// TIA Portal project "Bloques_y_Lenguajes" (V15)

(* hardware
DEVICE "S7-1200 station_1"  S7-1200 Station
   slot 0: "Rack_0"  S7-1200 Rack  Rack  V1.0
   slot 1: "PLC_1"  CPU 1215C DC/DC/DC  6ES7 215-1AG40-0XB0  V4.2
*)

// ===== PLC "PLC_1"  CPU 1215C DC/DC/DC =====

VAR_GLOBAL   // PLC tag table "Tabla de variables estándar"
   "MarcaTemperatura" AT %MD0 : Real;
   "Temperatura" AT %MD4 : Real;
   "Probabilidad_Temperatura" AT %MD8 : Real;
   "Presion" AT %MD12 : Real;
   "Probabilidad_Presion" AT %MD16 : Real;
   "Indicador_anomalia" AT %M20.0 : Bool;
   "Epsilon" AT %MD22 : Real;
   "Probabilidad_combinada" AT %MD26 : Real;
END_VAR

DATA_BLOCK "Variables1"   // DB1
{ S7_Optimized_Access := 'TRUE' }
VERSION : 0.1
   VAR
      Temperatura : Array[0..3600] of Real;
   END_VAR
   VAR RETAIN
      Puntero : Int := 1;
   END_VAR
   VAR
      Inyectora : Struct
         Temperatura : Struct
            Zona1 : Real;
            Zona2 : Real;
            Zona3 : Real;
            Zona4 : Real;
         END_STRUCT;
         Estado : Bool;
         Alarma : Bool;
      END_STRUCT;
   END_VAR
BEGIN
   Temperatura[5] := 235.87;
END_DATA_BLOCK

FUNCTION "Bloque_SCL" : Void   // FC1, SCL
{ S7_Optimized_Access := 'TRUE' }
VERSION : 0.1
BEGIN
   "MarcaTemperatura" := "Variables1".Temperatura["Variables1".Puntero];
END_FUNCTION

FUNCTION "Calacular_probabilidad_normal_temp" : Void   // FC2, SCL
{ S7_Optimized_Access := 'TRUE' }
VERSION : 0.1
   VAR_INPUT
      Media : Real;
      Desviacion_estandar : Real;
      Nuevo_Dato : Real;
   END_VAR
   VAR_OUTPUT
      Probabilidad : Real;
   END_VAR
   VAR CONSTANT
      Pi : Real := 3.1416;
   END_VAR
BEGIN
   #Probabilidad := EXP(-0.5 * SQR((#Nuevo_Dato - #Media) / #Desviacion_estandar))/((#Desviacion_estandar * SQRT(2.0*#Pi)));
END_FUNCTION

FUNCTION "Detector_de_anamolia" : Void   // FC3, SCL
{ S7_Optimized_Access := 'TRUE' }
VERSION : 0.1
   VAR_INPUT
      Probabilidad1 : Real;
      Probabilidad2 : Real;
      Epsilon : Real;
   END_VAR
   VAR_OUTPUT
      Indicacion_anomalia : Bool;
      "V alorProbabilidad_combinada" : Real;
   END_VAR
BEGIN
   IF #Probabilidad1 * #Probabilidad2 > #Epsilon  THEN
       #Indicacion_anomalia:=FALSE
       ;
   END_IF;

   IF #Probabilidad1 * #Probabilidad2 < #Epsilon THEN
       #Indicacion_anomalia:=TRUE
       ;
   END_IF;

   #"V alorProbabilidad_combinada" := #Probabilidad1 * #Probabilidad2;
END_FUNCTION

FUNCTION "Calcular_probabilidad_normal_presion" : Void   // FC4, SCL
{ S7_Optimized_Access := 'TRUE' }
VERSION : 0.1
   VAR_INPUT
      Media1 : Real;
      Desviacion_estandar1 : Real;
      Nuevo_Dato1 : Real;
   END_VAR
   VAR_OUTPUT
      Probabilidad1 : Real;
   END_VAR
   VAR CONSTANT
      Pi1 : Real := 3.1416;
   END_VAR
BEGIN
   #Probabilidad1 := EXP(-0.5 * SQR((#Nuevo_Dato1 - #Media1) / #Desviacion_estandar1)) / ((#Desviacion_estandar1 * SQRT(2.0 * #Pi1)));
END_FUNCTION

ORGANIZATION_BLOCK "Main"   // OB1, LAD, ProgramCycle
TITLE = "Main Program Sweep (Cycle)"
{ S7_Optimized_Access := 'TRUE' }
VERSION : 0.1
   VAR_INPUT
      Initial_Call : Bool;   // Initial call of this OB
      Remanence : Bool;   // =True, if remanent data are available
   END_VAR
BEGIN

REGION Network 1
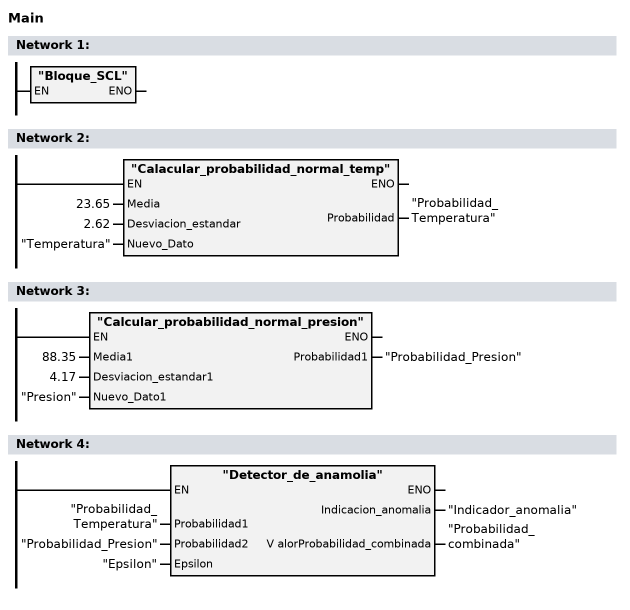
   RUNG wire#powerrail
      "Bloque_SCL"()
   END_RUNG
   // the same network as SCL:
   "Bloque_SCL"();
END_REGION

REGION Network 2
   RUNG wire#powerrail
      "Calacular_probabilidad_normal_temp"(Media := 23.65, Desviacion_estandar := 2.62, Nuevo_Dato := "Temperatura", Probabilidad => "Probabilidad_Temperatura")
   END_RUNG
   // the same network as SCL:
   "Calacular_probabilidad_normal_temp"(Media := 23.65,
                           Desviacion_estandar := 2.62,
                           Nuevo_Dato := "Temperatura",
                           Probabilidad => "Probabilidad_Temperatura");
END_REGION

REGION Network 3
   RUNG wire#powerrail
      "Calcular_probabilidad_normal_presion"(Media1 := 88.35, Desviacion_estandar1 := 4.17, Nuevo_Dato1 := "Presion", Probabilidad1 => "Probabilidad_Presion")
   END_RUNG
   // the same network as SCL:
   "Calcular_probabilidad_normal_presion"(Media1 := 88.35,
                           Desviacion_estandar1 := 4.17,
                           Nuevo_Dato1 := "Presion",
                           Probabilidad1 => "Probabilidad_Presion");
END_REGION

REGION Network 4
   RUNG wire#powerrail
      "Detector_de_anamolia"(Probabilidad1 := "Probabilidad_Temperatura", Probabilidad2 := "Probabilidad_Presion", Epsilon := "Epsilon", Indicacion_anomalia => "Indicador_anomalia", "V alorProbabilidad_combinada" => "Probabilidad_combinada")
   END_RUNG
   // the same network as SCL:
   "Detector_de_anamolia"(Probabilidad1 := "Probabilidad_Temperatura",
                          Probabilidad2 := "Probabilidad_Presion",
                          Epsilon := "Epsilon",
                          Indicacion_anomalia => "Indicador_anomalia",
                          "V alorProbabilidad_combinada" => "Probabilidad_combinada");
END_REGION
END_ORGANIZATION_BLOCK